// TwinCAT 3 PLC project ProcessSubElements
// Title: Process Sub-Elements
// Company: AnkerAndersen A/S
// Author: Benjamin Nielsen
// ProjectVersion: 1.0.0
// Description: Process Sub-Elements to be used in Process Elements
// ProgramVersion: 3.1.4026.1+972e9c44872ad038b353624a861fd7e3244e9f75
// libraries:
//   Tc2_Standard, * (Beckhoff Automation GmbH)
//   Tc2_System, * (Beckhoff Automation GmbH)
// project tree:
//   DUTs/ E_InverterState.TcDUT, E_State.TcDUT
//   / PlcTask.TcTTO
//   POUs/ FB_DigitalInput.TcPOU, FB_DigitalOutput.TcPOU, FB_Encoder.TcPOU, FB_Inverter.TcPOU, MAIN.TcPOU
//   Version/ Global_Version.TcGVL
// real-time tasks:
//   TASK PlcTask: cycle T#10ms, priority 20, ADS port 350

CONFIGURATION ProcessSubElements
    RESOURCE PLC ON TwinCAT3
        TASK PlcTask(INTERVAL := T#10ms, PRIORITY := 20);
        PROGRAM MAIN WITH PlcTask : MAIN;
    END_RESOURCE
END_CONFIGURATION

// ---- DUTs/E_InverterState.TcDUT
{attribute 'qualified_only'}
{attribute 'strict'}
TYPE E_InverterState :
(
	Stopped 	:= 0,
	Starting 	:= 1,
	Started 	:= 2,
	Paused		:= 3,
	Stopping	:= 4,
	Alarm		:= 5
);
END_TYPE

// ---- DUTs/E_State.TcDUT
{attribute 'qualified_only'}
{attribute 'strict'}
TYPE E_State :
(
	NormalOperation := 0,
	Simulation		:= 1,
	ConfigMode		:= 2
);
END_TYPE

// ---- Version/Global_Version.TcGVL
{attribute 'TcGenerated'}
{attribute 'no-analysis'}
{attribute 'linkalways'}
// This function has been automatically generated from the project information.
VAR_GLOBAL CONSTANT
	{attribute 'const_non_replaced'}
	stLibVersion_Process_Sub_Elements : ST_LibVersion := (iMajor := 1, iMinor := 0, iBuild := 0, iRevision := 0, nFlags := 0, sVersion := '1.0.0');
END_VAR

// ---- POUs/MAIN.TcPOU
PROGRAM MAIN
VAR
END_VAR

END_PROGRAM

// ---- POUs/FB_DigitalInput.TcPOU
FUNCTION_BLOCK FB_DigitalInput
VAR_INPUT
	eMachineState	:REFERENCE TO E_State;			//Normal Operation, Simulation, Config Mode.
	bSignalIn_IO	AT %I*: BOOL; 					//IO Signal 
	bSimulateIn		:BOOL;							//Simulated signal from program/HMI
	tOnDelayIn		:TIME;							//On delay time from HMI
	tOffDelayIn		:TIME;							//Off delay time from HMI
END_VAR
VAR_OUTPUT
	bSignalRawOut	:BOOL;							//Output signal without delay
	bSignalDelayOut	:BOOL;							//Output signal with delay
END_VAR
VAR
	TONDelayOn		:TON;							//Time on delay
	TOFDelayOff		:TOF;							//Time off delay
	tOnDelay		:TIME;							//Time set to on delay
	tOffDelay		:TIME;							//Time set to off delay
END_VAR

CASE eMachineState OF
	E_State.NormalOperation:
	
		//If no time delays are specified, send signal out equal to signal in. 
		IF tOnDelay = T#0S AND tOffDelay = T#0S THEN
			bSignalRawOut := bSignalIn_IO;
		ELSE
			//If time delays are specified, send signal out as delayed signal in.
			TONDelayOn(IN:=bSignalIn_IO, PT:=tOnDelay);
			TOFDelayOff(IN:=TONDelayOn.Q, PT:=tOffDelay);
			bSignalDelayOut := TONDelayOn.Q OR TOFDelayOff.Q;
		END_IF
		
	E_State.Simulation:
	
		//If no time delays are specified, send simulated signal out equal to simulated signal in. 
		IF tOnDelay = T#0S AND tOffDelay = T#0S THEN
			bSignalRawOut := bSimulateIn;
		ELSE
			//If time delays are specified, send simulated signal out as delayed simulated signal in.
			TONDelayOn(IN:=bSimulateIn, PT:=tOnDelay);
			TOFDelayOff(IN:=TONDelayOn.Q, PT:=tOffDelay);
			bSignalDelayOut := TONDelayOn.Q OR TOFDelayOff.Q;
		END_IF
		
	E_State.ConfigMode:
	
		//Set delay times when machine is in config.
		tOnDelay := tOnDelayIn;
		tOffDelay := tOffDelayIn;
END_CASE

END_FUNCTION_BLOCK

// ---- POUs/FB_DigitalOutput.TcPOU
FUNCTION_BLOCK FB_DigitalOutput
VAR_INPUT
	eMachineState	:REFERENCE TO E_State;			//Normal Operation, Simulation, Config Mode.
	bSignalIn		:BOOL; 							//Signal from program
	bSimulateIn		:BOOL;							//Simulated signal from program/HMI
	tOnDelayIn		:TIME;							//On delay time from HMI
	tOffDelayIn		:TIME;							//Off delay time from HMI
END_VAR
VAR_OUTPUT
	bSignalOut_IO	AT %Q* 	:BOOL;					//IO Signal 
END_VAR
VAR
	TONDelayOn		:TON;							//Time on delay
	TOFDelayOff		:TOF;							//Time off delay
	tOnDelay		:TIME;							//Time set to on delay
	tOffDelay		:TIME;							//Time set to off delay
END_VAR

CASE eMachineState OF
	E_State.NormalOperation:
	
		//If no time delays are specified, send signal out equal to signal in. 
		IF tOnDelay = T#0S AND tOffDelay = T#0S THEN
			bSignalOut_IO := bSignalIn;
		ELSE
			//If time delays are specified, send signal out as delayed signal in.
			TONDelayOn(IN:=bSignalIn, PT:=tOnDelay);
			TOFDelayOff(IN:=TONDelayOn.Q, PT:=tOffDelay);
			bSignalOut_IO := TONDelayOn.Q OR TOFDelayOff.Q;
		END_IF
		
	E_State.Simulation:
	
		//If no time delays are specified, send simulated signal out equal to simulated signal in. 
		IF tOnDelay = T#0S AND tOffDelay = T#0S THEN
			bSignalOut_IO := bSimulateIn;
		ELSE
			//If time delays are specified, send simulated signal out as delayed simulated signal in.
			TONDelayOn(IN:=bSimulateIn, PT:=tOnDelay);
			TOFDelayOff(IN:=TONDelayOn.Q, PT:=tOffDelay);
			bSignalOut_IO := TONDelayOn.Q OR TOFDelayOff.Q;
		END_IF
		
	E_State.ConfigMode:
	
		//Set delay times when machine is in config.
		tOnDelay := tOnDelayIn;
		tOffDelay := tOffDelayIn;
END_CASE

END_FUNCTION_BLOCK

// ---- POUs/FB_Encoder.TcPOU
FUNCTION_BLOCK FB_Encoder
VAR_INPUT
END_VAR
VAR_OUTPUT
END_VAR
VAR
END_VAR

END_FUNCTION_BLOCK

// ---- POUs/FB_Inverter.TcPOU
FUNCTION_BLOCK FB_Inverter
VAR_INPUT
END_VAR
VAR_OUTPUT
END_VAR
VAR
END_VAR

END_FUNCTION_BLOCK
